Staubli VAL3: OnF2.pgx

program OnF2()
begin
  call Edit()
end
